// Mitsubishi GX Works2 project: 서보 모터 위치 저장(기초)   PLC: Q03UDV

PROGRAM MAIN
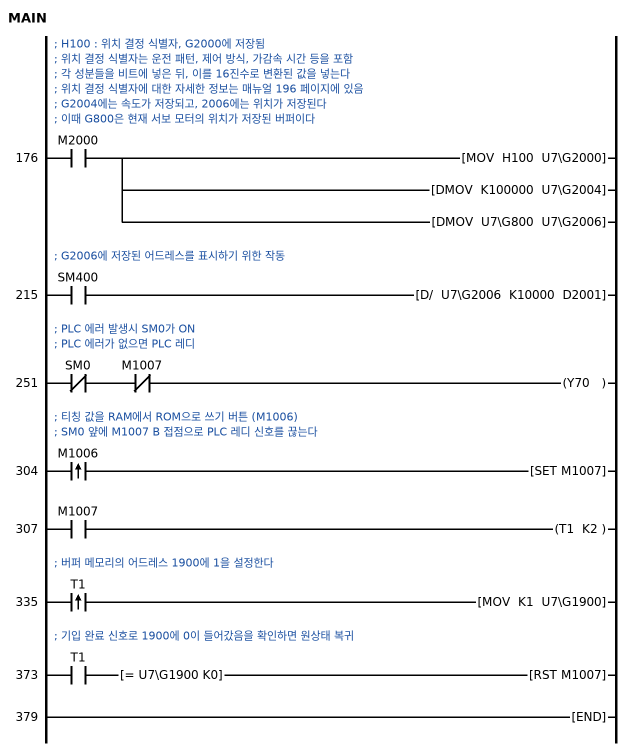
; H100 : 위치 결정 식별자, G2000에 저장됨
; 위치 결정 식별자는 운전 패턴, 제어 방식, 가감속 시간 등을 포함
; 각 성분들을 비트에 넣은 뒤, 이를 16진수로 변환된 값을 넣는다
; 위치 결정 식별자에 대한 자세한 정보는 매뉴얼 196 페이지에 있음
; G2004에는 속도가 저장되고, 2006에는 위치가 저장된다
; 이때 G800은 현재 서보 모터의 위치가 저장된 버퍼이다
176   LD      M2000
      MOV     H100 U7\G2000
      DMOV    K100000 U7\G2004
      DMOV    U7\G800 U7\G2006
; G2006에 저장된 어드레스를 표시하기 위한 작동
215   LD      SM400
      D/      U7\G2006 K10000 D2001
; PLC 에러 발생시 SM0가 ON
; PLC 에러가 없으면 PLC 레디
251   LDI     SM0
      ANI     M1007
      OUT     Y70
; 티칭 값을 RAM에서 ROM으로 쓰기 버튼 (M1006)
; SM0 얖에 M1007 B 접점으로 PLC 레디 신호를 끊는다
304   LDP     M1006
      SET     M1007
307   LD      M1007
      OUT     T1 K2
; 버퍼 메모리의 어드레스 1900에 1을 설정한다
335   LDP     T1
      MOV     K1 U7\G1900
; 기입 완료 신호로 1900에 0이 들어갔음을 확인하면 원상태 복귀
373   LD      T1
      AND=    U7\G1900 K0
      RST     M1007
379   END
END_PROGRAM
